// TwinCAT 3 PLC project Control_Monitor
// ProgramVersion: 3.1.4022.7
// libraries:
//   Tc2_ModbusSrv, * (Beckhoff Automation GmbH)
//   Tc2_Standard, * (Beckhoff Automation GmbH)
//   Tc2_System, * (Beckhoff Automation GmbH)
//   Tc3_Module, * (Beckhoff Automation GmbH)
//   VisuSymbols, * (System)
// project tree:
//   / GlobalTextList.TcGTLO, PlcTask.TcTTO, Visualization Manager.TcVMO (not stored)
//   GVLs/ Communication.TcGVL, Variables.TcGVL
//   POUs/ COMM_CISS.TcPOU, Display.TcPOU, Half_Rotation.TcPOU, Input_Mapping.TcPOU, MAIN.TcPOU, Output_Mapping.TcPOU, Blade_Control.TcPOU, SELECT.TcPOU
//   VISUs/ PaintVisualization.TcVIS
// real-time tasks:
//   TASK PlcTask: cycle T#10ms, priority 20, ADS port 350

CONFIGURATION Control_Monitor
    RESOURCE PLC ON TwinCAT3
        TASK PlcTask(INTERVAL := T#10ms, PRIORITY := 20);
        PROGRAM MAIN WITH PlcTask : MAIN;
        PROGRAM Input_Mapping WITH PlcTask : Input_Mapping;
        PROGRAM Output_Mapping WITH PlcTask : Output_Mapping;
        PROGRAM Display WITH PlcTask : Display;
        PROGRAM Blade_Control WITH PlcTask : Blade_Control;
        PROGRAM SELECT WITH PlcTask : SELECT;
    END_RESOURCE
END_CONFIGURATION

// ---- GVLs/Communication.TcGVL
{attribute 'qualified_only'}
VAR_GLOBAL
	
	////////////////////////////// CISS Sensor ///////////////////////////////
	
	///////////////////	 Raw CISS Sensor Information  ////////////////////////
	
	arrACCData AT %I*      			: ARRAY [1..6] OF INT;
	arrGYRData AT %I*   			: ARRAY [1..6] OF INT;	
	arrMAGData AT %I*     			: ARRAY [1..6] OF INT;		
	arrTEMPData AT %I*     			: INT;
	arrHUMData AT %I*    			: INT;
	arrPRESData AT %I*     			: INT;
	arrLIGHTData AT %I*       		: INT;
	arrNOISEData AT %I*        		: INT;

		
	/////////////////////////////////////////////////////////////////////////	



END_VAR

// ---- GVLs/Variables.TcGVL
{attribute 'qualified_only'}
VAR_GLOBAL
	
	///////////////////////////////////////// ROBOT CONTROLLER /////////////////////////////////////////

	(* Robot IO Signals *)

		(* Robot Physical Signals *)
	
			(* Robot Physical Digital Inputs *)	
		
				{attribute 'OPC.UA.DA' := '1'}
				bRobotReadyForNext AT %I*: BOOL := FALSE;
			
			(* End of Robot Physical Digital Inputs *)	
			
			(* Robot Physical Digital Outputs *)	
			
				{attribute 'OPC.UA.DA' := '1'}
				bSetRobotNextAction AT %Q* : BOOL := FALSE;
			
			(* End of Robot Physical Digital Outputs *)		
					
		(* End of Robot Physical Signals *)

		(* Robot Virtual Signals *)
		
			(* Robot Virtual Digital Inputs *)	
				
				{attribute 'OPC.UA.DA' := '1'}
				bIsRobotInPos AT %I* : BOOL; 
				
			(* End of Robot Virtual Digital Inputs *)
		
		(* End of Robot Virtual Signals *)
	
	(* End of Robot IO Signals *)
					
	///////////////////////////////////////// OMRON CONTROLLER /////////////////////////////////////////
	
	(* OMRON motor controller *)
		
		(* OMRON Physical Signals *)
	
			(* OMRON Digital Inputs *)
			
				{attribute 'OPC.UA.DA' := '1'}
				bIsOmronHome AT %I* : BOOL; (* Variable to start/stop signal reading *)
				
				{attribute 'OPC.UA.DA' := '1'}
				bIs_In_Pos AT %I* : BOOL; (* Variable to start/stop signal reading *)
				
				{attribute 'OPC.UA.DA' := '1'}
				bReadyForNext AT %I* : BOOL; (* Variable to start/stop signal reading *)
				
				{attribute 'OPC.UA.DA' := '1'}
				bIsMotorMoving AT %I* : BOOL; (* Variable to start/stop signal reading *)
			
			(* End of OMRON Digital Inputs *)
			
			(* OMRON Digital Outputs *)
			
				{attribute 'OPC.UA.DA' := '1'}
				bStartOperation AT %Q* : BOOL;	
						
				{attribute 'OPC.UA.DA' := '1'}
				bM0 AT %Q* : BOOL;	
				
				{attribute 'OPC.UA.DA' := '1'}
				bM1 AT %Q* : BOOL;	
			
				{attribute 'OPC.UA.DA' := '1'}
				bM2 AT %Q* : BOOL;		
				
				{attribute 'OPC.UA.DA' := '1'}
				bStopOperations AT %Q* : BOOL;	
				
				{attribute 'OPC.UA.DA' := '1'}
				bGoHomeOmron AT %Q* : BOOL;			
			
			(* End of OMRON Digital Outputs *)
			
		(* End of OMRON Physical Signals *)
	
		(* OMRON Virtual Signals *)
		
			(* OMRON Virtual Digital Inputs *)	
				
					{attribute 'OPC.UA.DA' := '1'}
					bIsOmronInPos AT %I* : BOOL; 				 
				
			(* End of OMRON Virtual Digital Inputs *)
		
		(* End of OMRON Virtual Signals *)
		
	(* Display Variables *)	
	
		{attribute 'OPC.UA.DA' := '1'}
		bPaint AT %Q* : BOOL;	
			
		{attribute 'OPC.UA.DA' := '1'}
		bSwitchON AT %I* : BOOL := FALSE;	
		
	(* End of Display Variables *)
	
	
	//////////////////////////////////////// Digitalization Workscope /////////////////////////////////////////

	(* Allow collection and visualization of data *)
	
		{attribute 'OPC.UA.DA' := '1'}
		bStartStop AT %I* : BOOL; (* Variable to start/stop signal reading *)
	
	
	(* Robot #1 Variables *)
	
	(* Robot Target *)
	(* {attribute 'OPC.UA.DA.Access' := '1'} *)
	
	{attribute 'OPC.UA.DA' := '1'}	
	fRTx : LREAL;
	
	{attribute 'OPC.UA.DA' := '1'}
	fRTy : LREAL;
	
	{attribute 'OPC.UA.DA' := '1'}
	fRTz : LREAL;
	
	{attribute 'OPC.UA.DA' := '1'}
	fRTq1 : LREAL;
	
	{attribute 'OPC.UA.DA' := '1'}
	fRTq2 : LREAL;
	
	{attribute 'OPC.UA.DA' := '1'}
	fRTq3 : LREAL;
	
	{attribute 'OPC.UA.DA' := '1'}
	fRTq4 : LREAL;
	
	{attribute 'OPC.UA.DA' := '1'}
	fRTcfg1 : LREAL;
	
	{attribute 'OPC.UA.DA' := '1'}
	fRTcfg2 : LREAL;
	
	{attribute 'OPC.UA.DA' := '1'}
	fRTcfg3 : LREAL;
	
	{attribute 'OPC.UA.DA' := '1'}
	fRTcfg4 : LREAL;
	
	{attribute 'OPC.UA.DA' := '1'}
	fRText1 : LREAL;
	
	{attribute 'OPC.UA.DA' := '1'}
	fRText2 : LREAL;
	
	{attribute 'OPC.UA.DA' := '1'}
	fRText3 : LREAL;
	
	{attribute 'OPC.UA.DA' := '1'}
	fRText4 : LREAL;
	
	{attribute 'OPC.UA.DA' := '1'}
	fRText5 : LREAL;
	
	{attribute 'OPC.UA.DA' := '1'}
	fRText6 : LREAL;
		
	
	
	(* Axes *)
	(* {attribute 'OPC.UA.DA.Access' := '1'} *)
	
	{attribute 'OPC.UA.DA' := '1'}	
	fJT1 : LREAL;
	
	{attribute 'OPC.UA.DA' := '1'}
	fJT2 : LREAL;
	
	{attribute 'OPC.UA.DA' := '1'}
	fJT3 : LREAL;
	
	{attribute 'OPC.UA.DA' := '1'}
	fJT4 : LREAL;
	
	{attribute 'OPC.UA.DA' := '1'}
	fJT5 : LREAL;
	
	{attribute 'OPC.UA.DA' := '1'}
	fJT6 : LREAL;
	
	{attribute 'OPC.UA.DA' := '1'}	
	fJText1 : LREAL;
	
	{attribute 'OPC.UA.DA' := '1'}
	fJText2 : LREAL;
	
	{attribute 'OPC.UA.DA' := '1'}
	fJText3 : LREAL;
	
	{attribute 'OPC.UA.DA' := '1'}
	fJText4 : LREAL;
	
	{attribute 'OPC.UA.DA' := '1'}
	fJText5 : LREAL;
	
	{attribute 'OPC.UA.DA' := '1'}
	fJText6 : LREAL;
	
	(* Robot Status *)
	
	{attribute 'OPC.UA.DA' := '1'}
	sRSstatus : STRING;
	
	
	(* Work Object Info *)
	
	{attribute 'OPC.UA.DA' := '1'}
	bWDrobhold : BOOL;
	
	{attribute 'OPC.UA.DA' := '1'}
	bWDufprog : BOOL;
	
	{attribute 'OPC.UA.DA' := '1'}
	sWDufmec : STRING;
	
	{attribute 'OPC.UA.DA' := '1'}	
	fWDux : LREAL;
	
	{attribute 'OPC.UA.DA' := '1'}
	fWDuy : LREAL;
	
	{attribute 'OPC.UA.DA' := '1'}
	fWDuz : LREAL;
	
	{attribute 'OPC.UA.DA' := '1'}
	fWDuq1 : LREAL;
	
	{attribute 'OPC.UA.DA' := '1'}
	fWDuq2 : LREAL;
	
	{attribute 'OPC.UA.DA' := '1'}
	fWDuq3 : LREAL;
	
	{attribute 'OPC.UA.DA' := '1'}
	fWDuq4 : LREAL;
	
	{attribute 'OPC.UA.DA' := '1'}	
	fWDox : LREAL;
	
	{attribute 'OPC.UA.DA' := '1'}
	fWDoy : LREAL;
	
	{attribute 'OPC.UA.DA' := '1'}
	fWDoz : LREAL;
	
	{attribute 'OPC.UA.DA' := '1'}
	fWDoq1 : LREAL;
	
	{attribute 'OPC.UA.DA' := '1'}
	fWDoq2 : LREAL;
	
	{attribute 'OPC.UA.DA' := '1'}
	fWDoq3 : LREAL;
	
	{attribute 'OPC.UA.DA' := '1'}
	fWDoq4 : LREAL;
	
	
	(* Tool Info *)
	
	{attribute 'OPC.UA.DA' := '1'}
	bTDrobhold : BOOL;
	
	{attribute 'OPC.UA.DA' := '1'}
	fTDx : LREAL;
	
	{attribute 'OPC.UA.DA' := '1'}
	fTDy : LREAL;
	
	{attribute 'OPC.UA.DA' := '1'}	
	fTDz : LREAL;
	
	{attribute 'OPC.UA.DA' := '1'}
	fTDq1 : LREAL;
	
	{attribute 'OPC.UA.DA' := '1'}
	fTDq2 : LREAL;
	
	{attribute 'OPC.UA.DA' := '1'}
	fTDq3 : LREAL;
	
	{attribute 'OPC.UA.DA' := '1'}
	fTDq4 : LREAL;
	
	{attribute 'OPC.UA.DA' := '1'}
	fTDmass : LREAL;
	
	{attribute 'OPC.UA.DA' := '1'}
	fTDcogx : LREAL;
	
	{attribute 'OPC.UA.DA' := '1'}	
	fTDcogy : LREAL;
	
	{attribute 'OPC.UA.DA' := '1'}
	fTDcogz : LREAL;
	
	{attribute 'OPC.UA.DA' := '1'}
	fTDcogq1 : LREAL;
	
	{attribute 'OPC.UA.DA' := '1'}
	fTDcogq2 : LREAL;
	
	{attribute 'OPC.UA.DA' := '1'}
	fTDcogq3 : LREAL;
	
	{attribute 'OPC.UA.DA' := '1'}
	fTDcogq4 : LREAL;
	
	{attribute 'OPC.UA.DA' := '1'}
	fTDix : LREAL;
	
	{attribute 'OPC.UA.DA' := '1'}
	fTDiy : LREAL;
	
	{attribute 'OPC.UA.DA' := '1'}
	fTDiz : LREAL;
	
	
	(* Robot #1 Environment Variables *)
	
	
	(* Sensors *)
		
	{attribute 'OPC.UA.DA' := '1'}	
	fAccX : LREAL;
	
	{attribute 'OPC.UA.DA' := '1'}	
	fAccY : LREAL;
	
	{attribute 'OPC.UA.DA' := '1'}	
	fAccZ : LREAL;
	
	{attribute 'OPC.UA.DA' := '1'}	
	fGyrX : LREAL;
	
	{attribute 'OPC.UA.DA' := '1'}	
	fGyrY : LREAL;
	
	{attribute 'OPC.UA.DA' := '1'}	
	fGyrZ : LREAL;
	
	{attribute 'OPC.UA.DA' := '1'}	
	fMagX : LREAL;
	
	{attribute 'OPC.UA.DA' := '1'}	
	fMagY : LREAL;
	
	{attribute 'OPC.UA.DA' := '1'}	
	fMagZ : LREAL;
	
	{attribute 'OPC.UA.DA' := '1'}	
	fTemp : LREAL;
	
	{attribute 'OPC.UA.DA' := '1'}	
	fHum : LREAL;
	
	{attribute 'OPC.UA.DA' := '1'}	
	fPres : LREAL;
	
	{attribute 'OPC.UA.DA' := '1'}	
	fLight : LREAL;
	
	{attribute 'OPC.UA.DA' := '1'}	
	fNoise : LREAL;
	
	{attribute 'OPC.UA.DA' := '1'}	
	fPPM : LREAL;
	
	
		
END_VAR

// ---- POUs/MAIN.TcPOU
PROGRAM MAIN
VAR	

END_VAR


IF NOT Variables.bStartStop THEN
	
	Variables.fJT1 := 0;
	Variables.fJT2 := 0;
	Variables.fJT3 := 0;
	Variables.fJT4 := 0;
	Variables.fJT5 := 0;
	Variables.fJT6 := 0;
	
	Variables.fRTx := 0;
	Variables.fRTy := 0;
	Variables.fRTz := 0;	
	Variables.fRTq1 := 0;
	Variables.fRTq2 := 0;
	Variables.fRTq3 := 0;
	Variables.fRTq4 := 0;
	
	Variables.fTDmass := 0;
	Variables.fTDx := 0;
	Variables.fTDy := 0;
	Variables.fTDz := 0;
	Variables.fTDq1 := 0;
	Variables.fTDq2 := 0;
	Variables.fTDq3 := 0;
	Variables.fTDq4 := 0;
	
	Variables.fTDcogx := 0;
	Variables.fTDcogy := 0;
	Variables.fTDcogz := 0;
	Variables.fTDcogq1 := 0;
	Variables.fTDcogq2 := 0;
	Variables.fTDcogq3 := 0;
	Variables.fTDcogq4 := 0;
	
	Variables.fTDix := 0;
	Variables.fTDiy := 0;
	Variables.fTDiz := 0;
	
	
	Variables.fWDox := 0;
	Variables.fWDoy := 0;
	Variables.fWDoz := 0;
	Variables.fWDoq1 := 0;
	Variables.fWDoq2 := 0;
	Variables.fWDoq3 := 0;
	Variables.fWDoq4 := 0;
	
	Variables.fWDux := 0;
	Variables.fWDuy := 0;
	Variables.fWDuz := 0;
	Variables.fWDuq1 := 0;
	Variables.fWDuq2 := 0;
	Variables.fWDuq3 := 0;
	Variables.fWDuq4 := 0;
	
END_IF


COMM_CISS();

END_PROGRAM

// ---- POUs/COMM_CISS.TcPOU
{attribute 'qualified_only}
PROGRAM COMM_CISS
VAR
	FB1: FB_MBReadRegs;
	
	// IP address & Port of ModBUS Server //
	ipAddr         					: STRING(15) := 'localhost';
	iMBPort							: UINT := 502;
	
	// Function Blocks to extract robot information //
	// CISS Sensor Addresses and Array Sizes //
	
	nAddrrAccelerometer				: WORD := 100;	
	nAddrrGyroscope					: WORD := 106;
	nAddrrMagnetometer				: WORD := 112;	
	nAddrrTemperature				: WORD := 118;
	nAddrrHumidity					: WORD := 120;	
	nAddrrPressure					: WORD := 122;
	nAddrrLight						: WORD := 124;	
	nAddrrNoise						: WORD := 126;
	
	
	nQtyUnit						: WORD := 2;
	nQtyCart						: WORD := 3;
	nQtyRot							: WORD := 3;	
	nQtyMixed						: WORD := 6;
		
	
	// Blocks //
	
	// CISS Accelerometer information //	
	fbCISSAccelerometer				: FB_MBReadRegs;
	// CISS Gyroscpe information //	
	fbCISSGyroscope					: FB_MBReadRegs;
	// CISS Magnetometer information //	
	fbCISSMagnetometer				: FB_MBReadRegs;
	// CISS Temperature information //	
	fbCISSTemperature				: FB_MBReadRegs;
	// CISS Humidity information //		
	fbCISSHumidity					: FB_MBReadRegs;
	// CISS Pressure information //	
	fbCISSPressure					: FB_MBReadRegs;
	// CISS Light information //	
	fbCISSLight						: FB_MBReadRegs;
	// CISS Noise information //	
	fbCISSNoise						: FB_MBReadRegs;
	
		
	// Reading Register - FB //
	fbReadRegs						: FB_MBReadRegs;
	bReadRegs						: BOOL;
	bReadRegsBusy   				: BOOL;
	bReadRegsError  				: BOOL;
	nReadRegsErrorId        		: UDINT;	
	
	// Writing Register - FB //
	fbWriteRegs						: FB_MBWriteRegs;
	bWriteRegs						: BOOL;
	bWriteRegsBusy   				: BOOL;
	bWriteRegsError  				: BOOL;
	nWriteRegsErrorId        		: UDINT;	
	
	// Error Variables //
	bError1, bError2, bError3		: BOOL;
	nErrID1, nErrID2, nErrID3		: UDINT;
	cbRead1, cbRead2, cbRead3		: UDINT;
	
	// Timers //
	TONreaders						: TON;
	TONwriters						: TON;
	tRefresh						: TIME := T#0.5S;
	tGiveUp							: TIME := T#2S;	
	
END_VAR

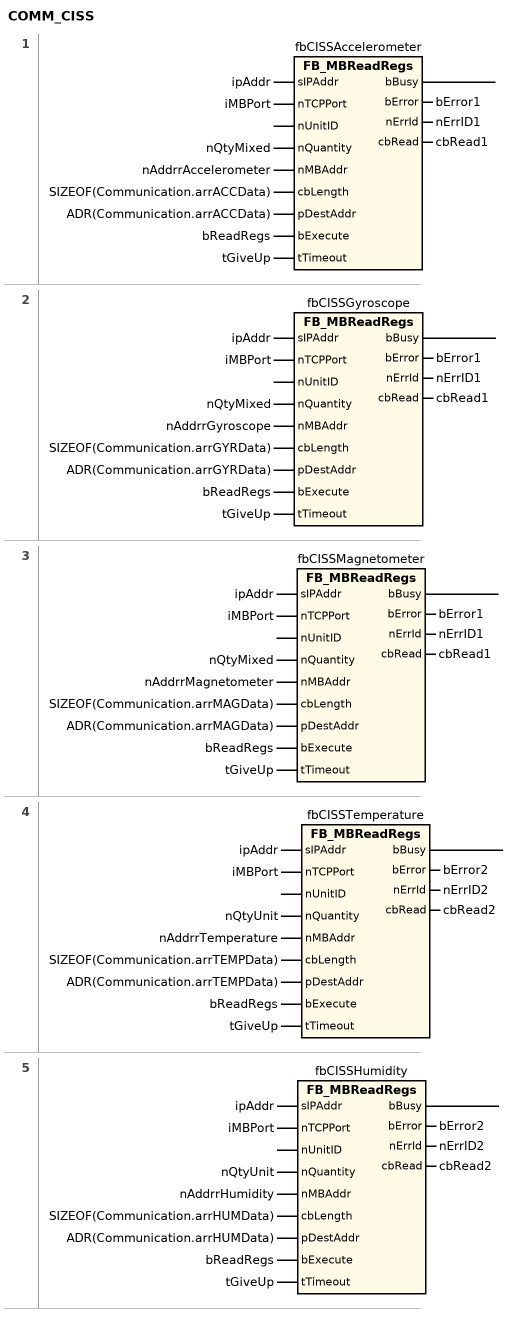
// NETWORK 1
fbCISSAccelerometer(
    sIPAddr := ipAddr,
    nTCPPort := iMBPort,
    nQuantity := nQtyMixed,
    nMBAddr := nAddrrAccelerometer,
    cbLength := SIZEOF(Communication.arrACCData),
    pDestAddr := ADR(Communication.arrACCData),
    bExecute := bReadRegs,
    tTimeout := tGiveUp,
    bError => bError1,
    nErrId => nErrID1,
    cbRead => cbRead1); // FB_MBReadRegs

// NETWORK 2
fbCISSGyroscope(
    sIPAddr := ipAddr,
    nTCPPort := iMBPort,
    nQuantity := nQtyMixed,
    nMBAddr := nAddrrGyroscope,
    cbLength := SIZEOF(Communication.arrGYRData),
    pDestAddr := ADR(Communication.arrGYRData),
    bExecute := bReadRegs,
    tTimeout := tGiveUp,
    bError => bError1,
    nErrId => nErrID1,
    cbRead => cbRead1); // FB_MBReadRegs

// NETWORK 3
fbCISSMagnetometer(
    sIPAddr := ipAddr,
    nTCPPort := iMBPort,
    nQuantity := nQtyMixed,
    nMBAddr := nAddrrMagnetometer,
    cbLength := SIZEOF(Communication.arrMAGData),
    pDestAddr := ADR(Communication.arrMAGData),
    bExecute := bReadRegs,
    tTimeout := tGiveUp,
    bError => bError1,
    nErrId => nErrID1,
    cbRead => cbRead1); // FB_MBReadRegs

// NETWORK 4
fbCISSTemperature(
    sIPAddr := ipAddr,
    nTCPPort := iMBPort,
    nQuantity := nQtyUnit,
    nMBAddr := nAddrrTemperature,
    cbLength := SIZEOF(Communication.arrTEMPData),
    pDestAddr := ADR(Communication.arrTEMPData),
    bExecute := bReadRegs,
    tTimeout := tGiveUp,
    bError => bError2,
    nErrId => nErrID2,
    cbRead => cbRead2); // FB_MBReadRegs

// NETWORK 5
fbCISSHumidity(
    sIPAddr := ipAddr,
    nTCPPort := iMBPort,
    nQuantity := nQtyUnit,
    nMBAddr := nAddrrHumidity,
    cbLength := SIZEOF(Communication.arrHUMData),
    pDestAddr := ADR(Communication.arrHUMData),
    bExecute := bReadRegs,
    tTimeout := tGiveUp,
    bError => bError2,
    nErrId => nErrID2,
    cbRead => cbRead2); // FB_MBReadRegs

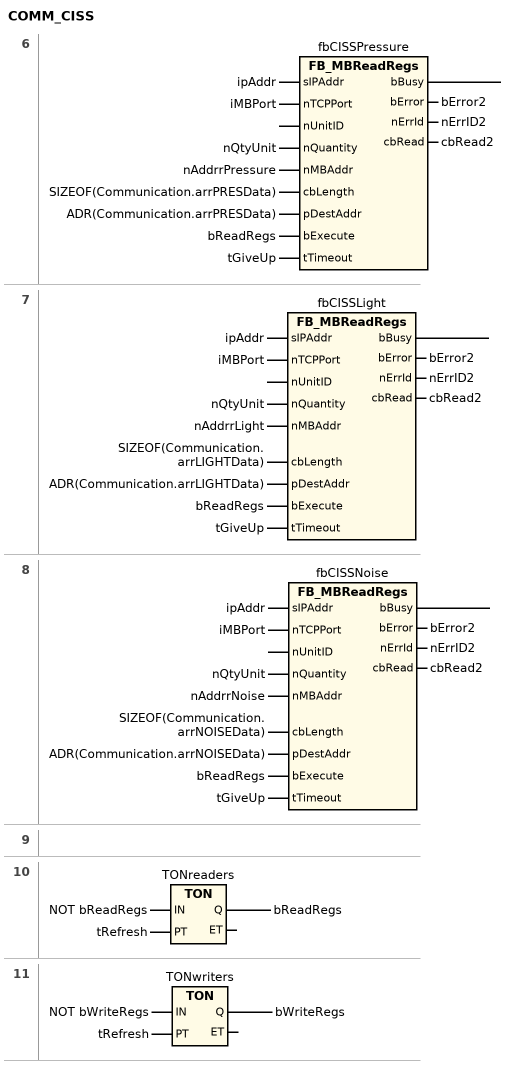
// NETWORK 6
fbCISSPressure(
    sIPAddr := ipAddr,
    nTCPPort := iMBPort,
    nQuantity := nQtyUnit,
    nMBAddr := nAddrrPressure,
    cbLength := SIZEOF(Communication.arrPRESData),
    pDestAddr := ADR(Communication.arrPRESData),
    bExecute := bReadRegs,
    tTimeout := tGiveUp,
    bError => bError2,
    nErrId => nErrID2,
    cbRead => cbRead2); // FB_MBReadRegs

// NETWORK 7
fbCISSLight(
    sIPAddr := ipAddr,
    nTCPPort := iMBPort,
    nQuantity := nQtyUnit,
    nMBAddr := nAddrrLight,
    cbLength := SIZEOF(Communication.arrLIGHTData),
    pDestAddr := ADR(Communication.arrLIGHTData),
    bExecute := bReadRegs,
    tTimeout := tGiveUp,
    bError => bError2,
    nErrId => nErrID2,
    cbRead => cbRead2); // FB_MBReadRegs

// NETWORK 8
fbCISSNoise(
    sIPAddr := ipAddr,
    nTCPPort := iMBPort,
    nQuantity := nQtyUnit,
    nMBAddr := nAddrrNoise,
    cbLength := SIZEOF(Communication.arrNOISEData),
    pDestAddr := ADR(Communication.arrNOISEData),
    bExecute := bReadRegs,
    tTimeout := tGiveUp,
    bError => bError2,
    nErrId => nErrID2,
    cbRead => cbRead2); // FB_MBReadRegs

// NETWORK 9

// NETWORK 10
TONreaders(IN := NOT bReadRegs, PT := tRefresh); // TON
bReadRegs := TONreaders.Q;

// NETWORK 11
TONwriters(IN := NOT bWriteRegs, PT := tRefresh); // TON
bWriteRegs := TONwriters.Q;

END_PROGRAM

// ---- POUs/Input_Mapping.TcPOU
PROGRAM Input_Mapping
VAR
	
END_VAR

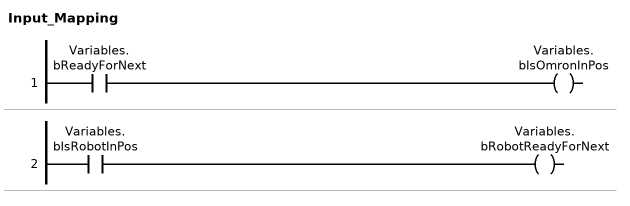
// NETWORK 1
Variables.bIsOmronInPos := Variables.bReadyForNext;

// NETWORK 2
Variables.bRobotReadyForNext := Variables.bIsRobotInPos;

END_PROGRAM

// ---- POUs/Output_Mapping.TcPOU
PROGRAM Output_Mapping
VAR
END_VAR

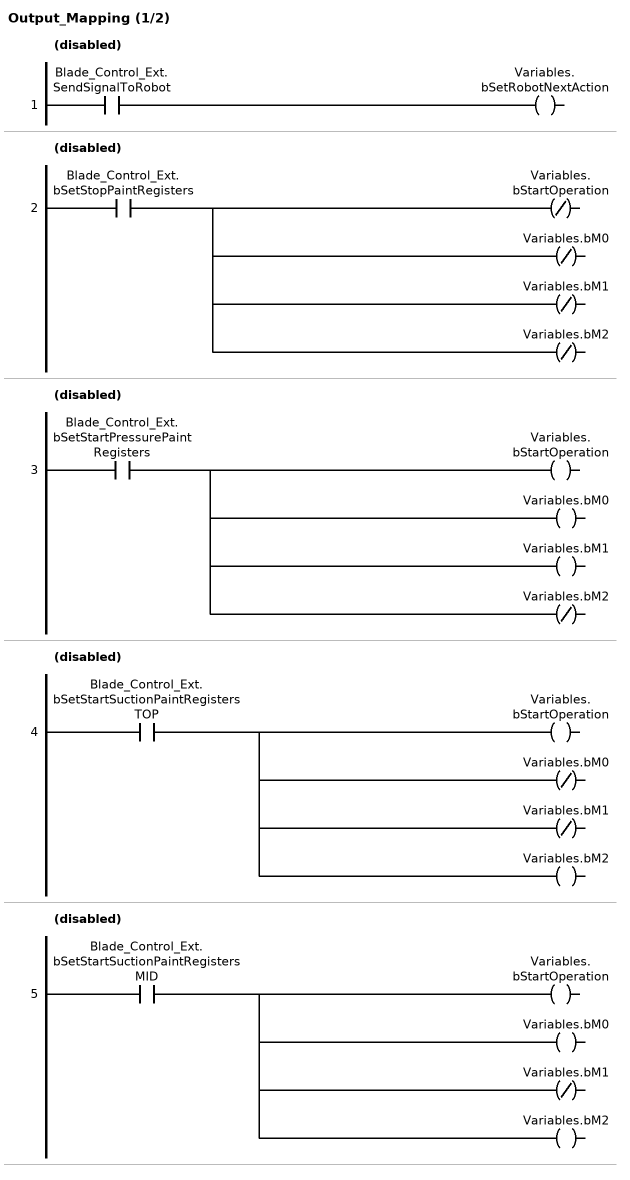
// NETWORK 1 (disabled)
// Variables.bSetRobotNextAction := Blade_Control_Ext.SendSignalToRobot;

// NETWORK 2 (disabled)
// Variables.bStartOperation := NOT Blade_Control_Ext.bSetStopPaintRegisters;
// Variables.bM0 := NOT Blade_Control_Ext.bSetStopPaintRegisters;
// Variables.bM1 := NOT Blade_Control_Ext.bSetStopPaintRegisters;
// Variables.bM2 := NOT Blade_Control_Ext.bSetStopPaintRegisters;

// NETWORK 3 (disabled)
// Variables.bStartOperation := Blade_Control_Ext.bSetStartPressurePaintRegisters;
// Variables.bM0 := Blade_Control_Ext.bSetStartPressurePaintRegisters;
// Variables.bM1 := Blade_Control_Ext.bSetStartPressurePaintRegisters;
// Variables.bM2 := NOT Blade_Control_Ext.bSetStartPressurePaintRegisters;

// NETWORK 4 (disabled)
// Variables.bStartOperation := Blade_Control_Ext.bSetStartSuctionPaintRegistersTOP;
// Variables.bM0 := NOT Blade_Control_Ext.bSetStartSuctionPaintRegistersTOP;
// Variables.bM1 := NOT Blade_Control_Ext.bSetStartSuctionPaintRegistersTOP;
// Variables.bM2 := Blade_Control_Ext.bSetStartSuctionPaintRegistersTOP;

// NETWORK 5 (disabled)
// Variables.bStartOperation := Blade_Control_Ext.bSetStartSuctionPaintRegistersMID;
// Variables.bM0 := Blade_Control_Ext.bSetStartSuctionPaintRegistersMID;
// Variables.bM1 := NOT Blade_Control_Ext.bSetStartSuctionPaintRegistersMID;
// Variables.bM2 := Blade_Control_Ext.bSetStartSuctionPaintRegistersMID;

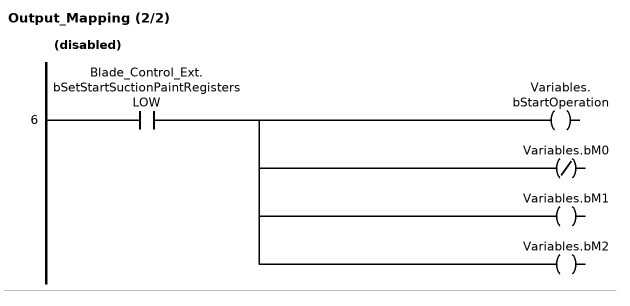
// NETWORK 6 (disabled)
// Variables.bStartOperation := Blade_Control_Ext.bSetStartSuctionPaintRegistersLOW;
// Variables.bM0 := NOT Blade_Control_Ext.bSetStartSuctionPaintRegistersLOW;
// Variables.bM1 := Blade_Control_Ext.bSetStartSuctionPaintRegistersLOW;
// Variables.bM2 := Blade_Control_Ext.bSetStartSuctionPaintRegistersLOW;

END_PROGRAM

// ---- POUs/Display.TcPOU
PROGRAM Display
VAR
	iDisplay_Value : UINT := 0;
	status_display : WSTRING;
	
	
	iDisplay_Component: INT;
	side_display	: WSTRING;
END_VAR

//Power Off Display
IF NOT Variables.bStartOperation THEN
	iDisplay_Value :=0;
END_IF;

//Power On Display
IF Variables.bStartOperation THEN
	iDisplay_Value :=1;
END_IF;

//Emergency Stop Display
IF Variables.bStopOperations THEN
	iDisplay_Value :=2;
END_IF;

//Painting Position Display
IF Variables.bIsOmronInPos THEN
	iDisplay_Value :=3;
END_IF;

//Painting Process Display
IF Variables.bPaint THEN
	iDisplay_Value :=4;
END_IF;

//Robotic Arm Movement Display
IF Variables.bIsRobotInPos THEN
	iDisplay_Value :=5;
END_IF;

//Process Completion Display
IF Half_Rotation.bProcess THEN
	iDisplay_Value :=6;
END_IF;

//Robotic Arm Movement Display
IF Half_Rotation.bRotation_Trig THEN
	iDisplay_Value :=7;
END_IF;

//Display Value to Display String (Process Type)
CASE iDisplay_Value OF
	
	0: status_display := "IDLE...";
	1: status_display := "POWER ON";
	2: status_display := "EMERGENCY STOP";
	3: status_display := "PAINT PROCESS READY";
	4: status_display := "PAINTING IN PROGRESS";
	5: status_display := "SHIFTING OF ROBOTIC ARM";
	6: status_display := "PAINT COMPLETED";
	7: status_display := "ROTATING SIDE";
	
END_CASE

//Display Value to Display String (Component Surface)
IF Half_Rotation.bFlip_Side THEN
	
	iDisplay_Component := 1;
	
	ELSE
		iDisplay_Component :=0;
END_IF


//Display for Component Surface Side
CASE iDisplay_Component OF
	
	0: side_display := "PRESSURE SIDE";
	1: side_display := "SUCTION SIDE";

END_CASE

END_PROGRAM

// ---- POUs/Half_Rotation.TcPOU
PROGRAM Half_Rotation
VAR
	bRotation_Trig : BOOL;
	bFlip_Side: BOOL;
	bProcess: BOOL;
END_VAR

END_PROGRAM

// ---- POUs/Blade_Control.TcPOU
PROGRAM Blade_Control
VAR
		{attribute 'OPC.UA.DA' := '1'}
	MY_TON : TON;
	MY_TON2: TON;
	MY_TON3: TON;
	MY_TON4: TON;
	MY_TON5: TON;
	
	SystemON: BOOL := FALSE;
	SystemReady: BOOL := FALSE;
	SendSignalToRobot: BOOL := FALSE;
	
	bSetStartPressurePaintRegisters: BOOL := FALSE;
	bSetStartSuctionPaintRegistersTOP: BOOL := FALSE; 
	bSetStartSuctionPaintRegistersMID: BOOL := FALSE; 
	bSetStartSuctionPaintRegistersLOW: BOOL := FALSE; 
	bSetStopPaintRegisters: BOOL := TRUE;
		
	Phase: INT := 0;	
	
	R1: BOOL := FALSE;	
	R2: BOOL := FALSE;
	R3: BOOL := FALSE;	
	R4: BOOL := FALSE;
	R5: BOOL := FALSE;		
	
	S1: BOOL := FALSE;
	S2: BOOL := FALSE;
	S3: BOOL := FALSE;

	
END_VAR
VAR // added by the converter: edge detectors and wires of the graphical bodies
    _w1, _w2, _w3, _w4, _w5, _w6, _w7, _w8, _w9, _w10, _w11, _w12, _w13, _w14, _w15 : BOOL;
END_VAR

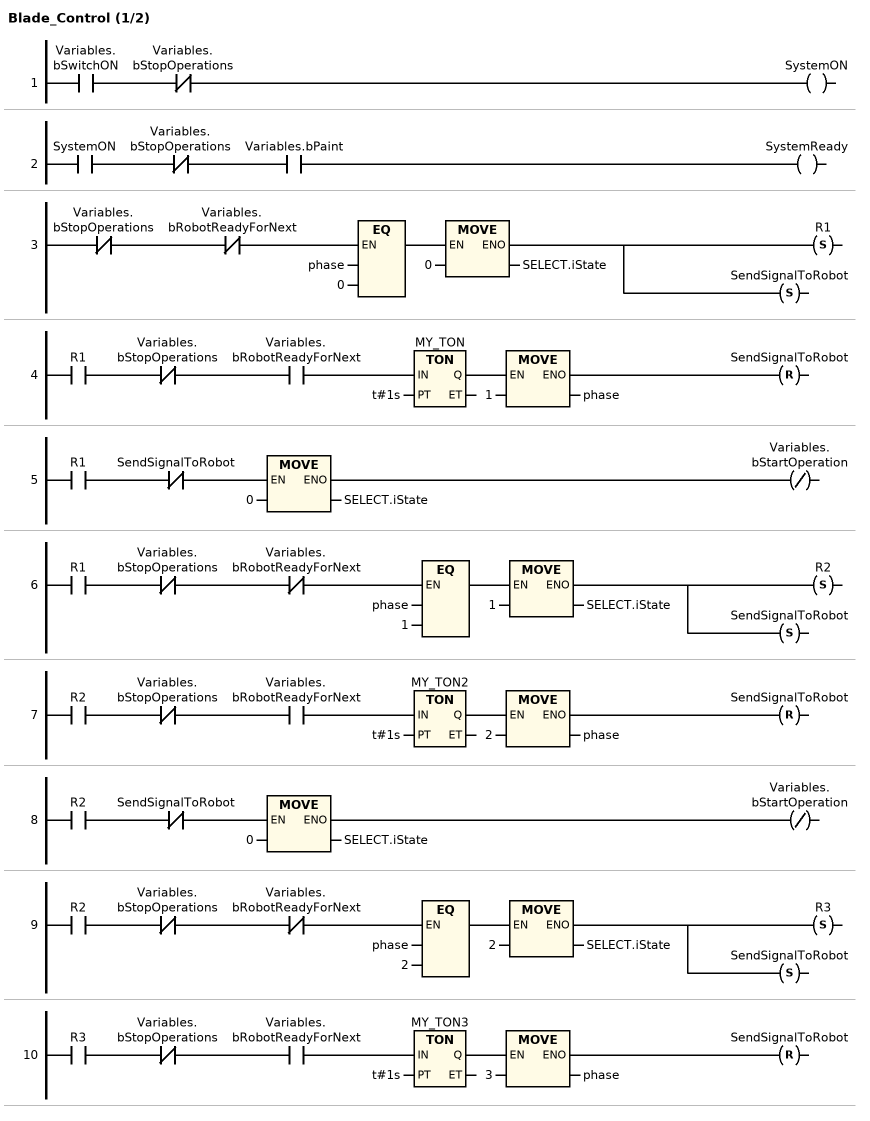
// NETWORK 1
SystemON := Variables.bSwitchON AND NOT Variables.bStopOperations;

// NETWORK 2
SystemReady := SystemON AND NOT Variables.bStopOperations AND Variables.bPaint;

// NETWORK 3
_w1 := NOT Variables.bStopOperations AND NOT Variables.bRobotReadyForNext AND phase = 0;
IF _w1 THEN SELECT.iState := 0; END_IF
R1 S= _w1;
SendSignalToRobot S= _w1;

// NETWORK 4
MY_TON(IN := R1 AND NOT Variables.bStopOperations AND Variables.bRobotReadyForNext, PT := t#1s); // TON
_w2 := MY_TON.Q;
IF _w2 THEN phase := 1; END_IF
SendSignalToRobot R= _w2;

// NETWORK 5
_w3 := R1 AND NOT SendSignalToRobot;
IF _w3 THEN SELECT.iState := 0; END_IF
Variables.bStartOperation := NOT _w3;

// NETWORK 6
_w4 := R1 AND NOT Variables.bStopOperations AND NOT Variables.bRobotReadyForNext AND phase = 1;
IF _w4 THEN SELECT.iState := 1; END_IF
R2 S= _w4;
SendSignalToRobot S= _w4;

// NETWORK 7
MY_TON2(IN := R2 AND NOT Variables.bStopOperations AND Variables.bRobotReadyForNext, PT := t#1s); // TON
_w5 := MY_TON2.Q;
IF _w5 THEN phase := 2; END_IF
SendSignalToRobot R= _w5;

// NETWORK 8
_w6 := R2 AND NOT SendSignalToRobot;
IF _w6 THEN SELECT.iState := 0; END_IF
Variables.bStartOperation := NOT _w6;

// NETWORK 9
_w7 := R2 AND NOT Variables.bStopOperations AND NOT Variables.bRobotReadyForNext AND phase = 2;
IF _w7 THEN SELECT.iState := 2; END_IF
R3 S= _w7;
SendSignalToRobot S= _w7;

// NETWORK 10
MY_TON3(IN := R3 AND NOT Variables.bStopOperations AND Variables.bRobotReadyForNext, PT := t#1s); // TON
_w8 := MY_TON3.Q;
IF _w8 THEN phase := 3; END_IF
SendSignalToRobot R= _w8;

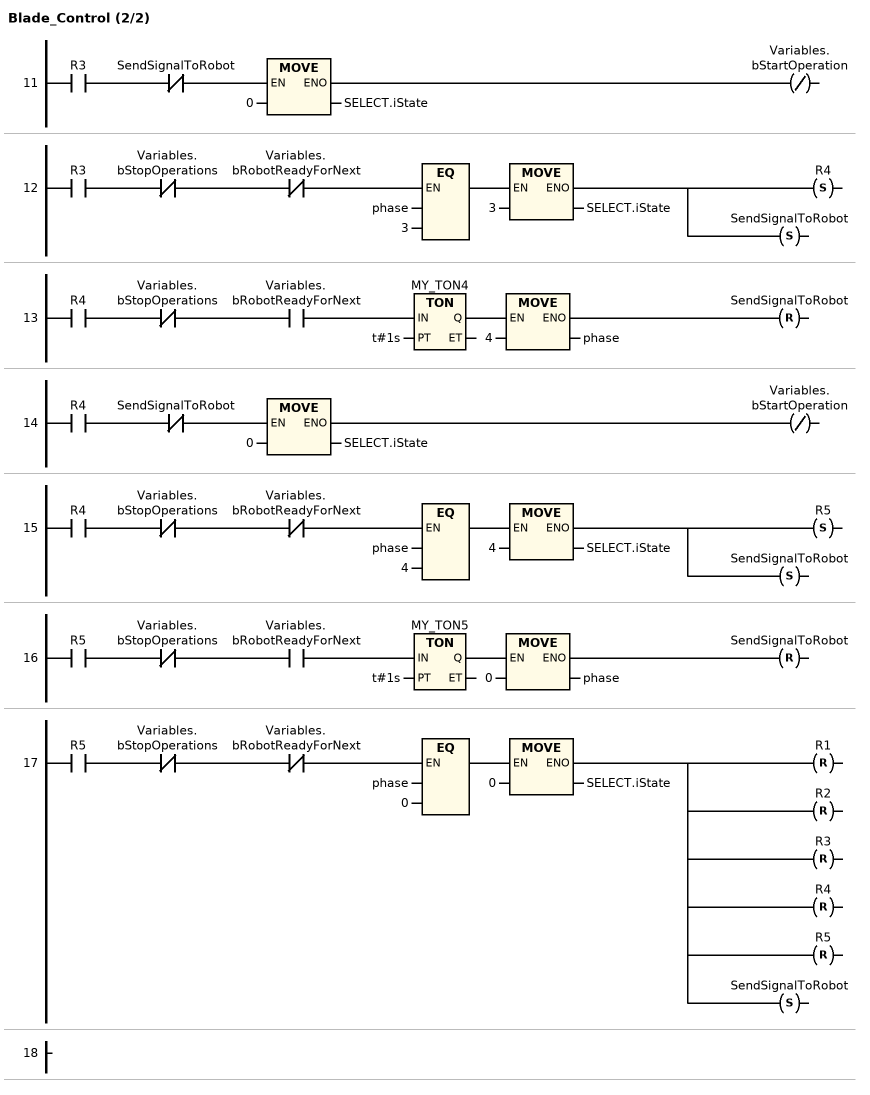
// NETWORK 11
_w9 := R3 AND NOT SendSignalToRobot;
IF _w9 THEN SELECT.iState := 0; END_IF
Variables.bStartOperation := NOT _w9;

// NETWORK 12
_w10 := R3 AND NOT Variables.bStopOperations AND NOT Variables.bRobotReadyForNext AND phase = 3;
IF _w10 THEN SELECT.iState := 3; END_IF
R4 S= _w10;
SendSignalToRobot S= _w10;

// NETWORK 13
MY_TON4(IN := R4 AND NOT Variables.bStopOperations AND Variables.bRobotReadyForNext, PT := t#1s); // TON
_w11 := MY_TON4.Q;
IF _w11 THEN phase := 4; END_IF
SendSignalToRobot R= _w11;

// NETWORK 14
_w12 := R4 AND NOT SendSignalToRobot;
IF _w12 THEN SELECT.iState := 0; END_IF
Variables.bStartOperation := NOT _w12;

// NETWORK 15
_w13 := R4 AND NOT Variables.bStopOperations AND NOT Variables.bRobotReadyForNext AND phase = 4;
IF _w13 THEN SELECT.iState := 4; END_IF
R5 S= _w13;
SendSignalToRobot S= _w13;

// NETWORK 16
MY_TON5(IN := R5 AND NOT Variables.bStopOperations AND Variables.bRobotReadyForNext, PT := t#1s); // TON
_w14 := MY_TON5.Q;
IF _w14 THEN phase := 0; END_IF
SendSignalToRobot R= _w14;

// NETWORK 17
_w15 := R5 AND NOT Variables.bStopOperations AND NOT Variables.bRobotReadyForNext AND phase = 0;
IF _w15 THEN SELECT.iState := 0; END_IF
R1 R= _w15;
R2 R= _w15;
R3 R= _w15;
R4 R= _w15;
R5 R= _w15;
SendSignalToRobot S= _w15;

// NETWORK 18

END_PROGRAM

// ---- POUs/SELECT.TcPOU
PROGRAM SELECT
VAR_INPUT
	iState AT %I*:	 INT := 0;
END_VAR
VAR
	bSwitch: BOOL := FALSE;
	WAIT1: TON;
	WAIT2: TON;
	WAIT3: TON;
	WAIT4: TON;
	
END_VAR


CASE iState OF

0: (* IDLE *)	
	Variables.bM0 := FALSE;
	Variables.bM1 := FALSE;
	Variables.bM2 := FALSE;
	Variables.bStartOperation := FALSE;
		
1: (* Pressure side *)	
	Variables.bM0 := FALSE;
	Variables.bM1 := TRUE;
	Variables.bM2 := FALSE;
	Variables.bStartOperation := TRUE;
	
2: (* Suction side Top *)
	Variables.bM0 := FALSE;
	Variables.bM1 := FALSE;
	Variables.bM2 := TRUE;
	Variables.bStartOperation := TRUE;

3: (* Suction side Mid *)
	Variables.bM0 := TRUE;
	Variables.bM1 := FALSE;
	Variables.bM2 := TRUE;
	Variables.bStartOperation := TRUE;

4: (* Suction side Bottom *)
	Variables.bM0 := FALSE;
	Variables.bM1 := TRUE;
	Variables.bM2 := TRUE;
	Variables.bStartOperation := TRUE;

END_CASE

END_PROGRAM

// ---- GlobalTextList.TcGTLO
TEXTLIST GlobalTextList
  368 = 'Initialize'
  230 = 'Is it in Position'
  293 = 'Motor off'
  957 = 'Moving?'
  381 = 'Omron OK Pos?'
  566 = 'Omron reached Position?'
  27 = 'Paint'
  846 = 'Painting'
  866 = 'Painting Process'
  191 = 'Painting?'
  544 = 'Power'
  997 = 'Reached Position'
  966 = 'Reached Position?'
  360 = 'Robot OK Pos?'
  0 = 'Robot Sim'
  217 = 'Start'
  168 = 'Status Display'
  32 = 'Stop'
END_TEXTLIST

// ---- VISUs/PaintVisualization.TcVIS
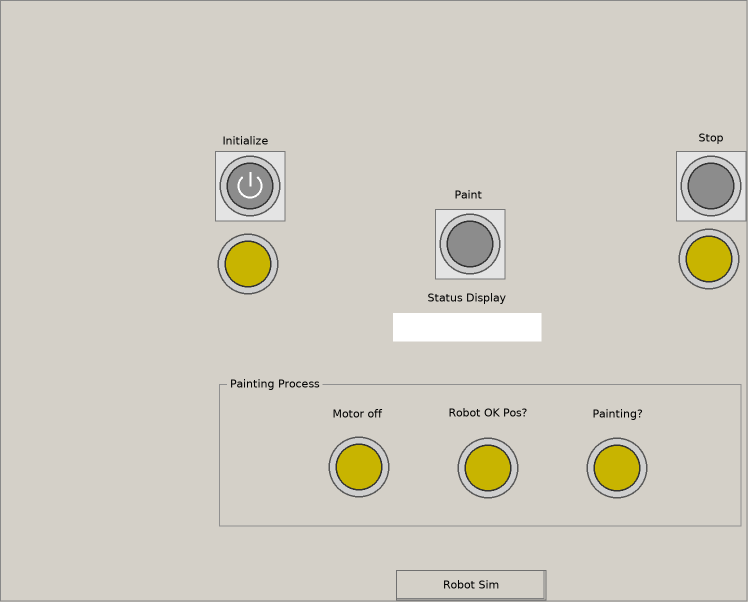
VISUALIZATION PaintVisualization  // 748x602
    GroupBox (219,376 522x150), "Painting Process"
        Label (92,18 93x40), "Motor off"
        Label (195,17 148x40), "Robot OK Pos?"
        Lamp1 (234,57 70x70), variable: Variables.bIsRobotInPos, style: Lamp-Lamp1-Yellow
        Lamp1 (105,56 70x70), style: Lamp-Lamp1-Yellow
    Lamp1 (213,229 70x70), variable: Variables.bSwitchON, style: Lamp-Lamp1-Yellow
    PushSwitch (676,151 70x70), variable: Variables.bStopOperations, behaviour: TOGGLE, style: Switch-PushSwitch-Gray
    Label (213,126 65x30), "Initialize"
    Label (685,123 52x30), "Stop"
    Lamp1 (582,433 70x70), style: Lamp-Lamp1-Yellow
    Label (541,399 154x30), "Painting?"
    PushSwitchLed (435,209 70x70), variable: Variables.bPaint, behaviour: TOGGLE, style: Switch-PushSwitchLed-Gray
    Label (436,180 65x30), "Paint"
    Textfield (392,312 150x30), text variable: Display.status_display
    Label (392,283 150x30), "Status Display"
    Lamp1 (674,224 70x70), variable: Variables.bStopOperations, style: Lamp-Lamp1-Yellow
    PowerSwitch (215,151 70x70), variable: Variables.bSwitchON, behaviour: TOGGLE, style: Switch-PowerSwitch-Gray
    Button (396,570 150x30), "Robot Sim"
        tap Variables.bIsRobotInPos
END_VISUALIZATION
